{attribute 'GeneratedUsingTerminal: EPP3744-0041-0016'}
{attribute addProperty BoxType "EPP3744-0041-0016"}
{attribute addProperty Id "InputAT %I*ARRAY[0..5] OF BOOL6"}
{attribute addProperty CRC "390650255"}
{attribute addProperty Size "6"}
TYPE DIG_Inputs_697E0EF2 EXTENDS InputBase_8311D824 :
STRUCT
	{attribute addProperty Name "Input"}
	Input AT %I* : ARRAY[0..5] OF BOOL;
END_STRUCT
END_TYPE

(* stored: Version 1.2.0.0, ProductVersion 3.1.4024.9
   DUT DIG_Inputs_697E0EF2: Id {0958c2f3-c069-435b-ac4d-c43b05e2d278} *)
